FUNCTION_BLOCK FB_Example
VAR
    iValue : INT;
END_VAR
BEGIN
iResult := iValue + 1;
END_FUNCTION_BLOCK
